FUNCTION F_Dewpoint : REAL
VAR_INPUT
	// relative humidity
	relhum:	REAL;
	// temperature °C
	t: REAL;
END_VAR
VAR
	a, b, 
	// Sättigungsdampfdruck in hPa
	sdd, 
	// Dampfdruck in hPa
	dd, v: REAL;
END_VAR

// source https://www.wetterochs.de/wetter/feuchte.html
IF t < 0.0 THEN
	a := 7.6; b := 240.7;// für T < 0 über Wasser (Taupunkt)
ELSE
	a := 7.5; b := 237.3;
END_IF

F_Dewpoint := -273.15;
IF b+T > 0 THEN
	SDD := LREAL_TO_REAL(6.1078 * EXPT(10, (a*T)/(b+T)));
ELSE
	SDD := 6.1078;
END_IF

DD := relhum/100.0 * SDD;
v := LOG(DD/6.1078);
IF a <> v THEN
	F_Dewpoint := b*v/(a-v);	
END_IF

END_FUNCTION

(* stored: Version 1.1.0.1, ProductVersion 3.1.4024.9
   POU F_Dewpoint: Id {1075508b-0103-445e-af41-8392a971b7cf}, SpecialFunc None *)
